FUNCTION_BLOCK Task2
VAR_INPUT
END_VAR
VAR_OUTPUT
END_VAR
VAR
	
	axTest : ARRAY[0..19] OF BOOL;
	i	:INT;
	
END_VAR

FOR i := 0 TO 19 BY 1 DO 	
	axTest[i]:= FALSE;
END_FOR
axTest[7]:= TRUE;

CheckIfAnyArrayElementIsTrue(axCheckTest:=axTest);

METHOD CheckIfAnyArrayElementIsTrue : BOOL
VAR_INPUT
	axCheckTest : ARRAY[0..19] OF BOOL;
END_VAR
VAR
	i	:INT;
	xCheck:BOOL;
END_VAR
VAR_INST
	xInArrayExistsTrueValue:BOOL;
END_VAR
FOR i := 0 TO 19 BY 1 DO 		
	
	IF axCheckTest[i] THEN
		
		xInArrayExistsTrueValue:=TRUE;
	
	ELSE
		;
	END_IF
	
END_FOR
END_METHOD

END_FUNCTION_BLOCK

(* stored: Version 1.1.0.1, ProductVersion 3.1.4024.13
   POU Task2: Id {c7253e7e-121f-4445-82f2-1134c52642e9}, SpecialFunc None
   Method CheckIfAnyArrayElementIsTrue: Id {f7ef02a5-b49f-4830-9531-ce54502d9b61} *)
